PROGRAM MAIN
VAR
	Counter0Inc : DWORD := 1;
	Counter0Read : DWORD; 
	Counter0 : count_mgr_test;
	Encoder0Read : ULINT;
	Encoder0	:	ST_BisscEncoder;
	EncoderDemand0 : ST_BeamDemand;
END_VAR

Counter0(Increment:=Counter0Inc);
Counter0Read := Counter0.CurrentOut;
EncoderDemand0 := BisscEvaluator(Encoder0);

END_PROGRAM

(* stored: Version 1.1.0.1, ProductVersion 3.1.4020.12
   POU MAIN: Id {ee27c5ec-ece1-4706-a959-f409661eea2d}, SpecialFunc None *)
